{attribute 'qualified_only'}
{attribute 'strict'}
{attribute 'to_string'}
TYPE E_Direction :
(
	STOP := 0,
	UP := 1,
	DOWN := 2
);
END_TYPE

(* stored: Version 1.1.0.1, ProductVersion 3.1.4024.12
   DUT E_Direction: Id {819ec583-5655-4fbe-94e1-919759458a46} *)
